# EPICS substitutions: example/exampleApp/Db/example.substitutions
file ADSimPeaks.template
{
pattern {P, R, PORT, ADDR, TIMEOUT}
        {ST99:Det, :Det1:, D1.SIM, 0, 1}
}

file ADSimPeaksBackground.template
{
pattern {P, R, PORT, ADDR, TIMEOUT}
        {ST99:Det, :Det1:, D1.SIM, 0, 1}
}

file ADSimPeaksPeak.template
{
pattern {P, R, PORT, ADDR, TIMEOUT, PEAK}
        {ST99:Det, :Det1:, D1.SIM, 0, 1, 0}
	{ST99:Det, :Det1:, D1.SIM, 0, 1, 1}
	{ST99:Det, :Det1:, D1.SIM, 0, 1, 2}
	{ST99:Det, :Det1:, D1.SIM, 0, 1, 3}
	{ST99:Det, :Det1:, D1.SIM, 0, 1, 4}
	{ST99:Det, :Det1:, D1.SIM, 0, 1, 5}
	{ST99:Det, :Det1:, D1.SIM, 0, 1, 6}
	{ST99:Det, :Det1:, D1.SIM, 0, 1, 7}
}

file NDCodec.template
{
pattern {P, R, PORT, ADDR, TIMEOUT, NDARRAY_PORT, NDARRAY_ADDR}
        {ST99:Det, :Det1:CO1:, D1.CO1, 0, 1, D1.SIM, 0}
}

file NDPva.template
{
pattern {P, R, PORT, ADDR, TIMEOUT, NDARRAY_PORT, NDARRAY_ADDR}
        {ST99:Det, :Det1:PV1:, D1.PV1, 0, 1, D1.CO1, 0}
}

file save_restoreStatus.db
{
pattern {P}
        {ST99:Det:IOC_SADet1:}
}

file ioc_sns.db
{
pattern {IOCNAME}
        {ST99:Det:IOC_SIDet1}
}
